PROGRAM PRG_HMI
VAR
	

	tonCaseDelay				: ARRAY [1..20] OF TON;
	tofCase						: ARRAY [1..20] OF TOF;
	rtrigCaseTriger				: ARRAY [1..20] OF R_TRIG;

	tonResetStatistics			: TON;
	
	fbWritePersistentData		:FB_WritePersistentData;
	fWritePersistentData		: F_TRIG;
	
END_VAR

ACT_ScreensNamesSet();
ACT_Buttons();
ACT_TimTrig();
ACT_General();
ACT_SavePersistentVariables();

tonResetStatistics( IN := 	GVL_HMI_GLOBAL.aResetHeightSensorBadParts [1] 	OR
							GVL_HMI_GLOBAL.aResetHeightSensorBadParts [2] 	OR
							GVL_HMI_GLOBAL.aResetHeightSensorBadParts [3] 	OR
							GVL_HMI_GLOBAL.aResetHeightSensorBadParts [4] 	OR
							GVL_HMI_GLOBAL.aResetHeightSensorGoodParts[1]	OR
							GVL_HMI_GLOBAL.aResetHeightSensorGoodParts[2]	OR
							GVL_HMI_GLOBAL.aResetHeightSensorGoodParts[3]	OR
							GVL_HMI_GLOBAL.aResetHeightSensorGoodParts[4]	OR
							GVL_HMI_GLOBAL.bResetHeightFailParts			OR
							GVL_HMI_GLOBAL.bResetHeightGoodParts			OR
							GVL_HMI_GLOBAL.bResetGoodParts					OR
							GVL_HMI_GLOBAL.bResetVisionBadParts				OR
							GVL_HMI_GLOBAL.bResetVisionGoodParts			OR
							GVL_HMI_GLOBAL.bResetFailedParts				OR
							GVL_HMI_GLOBAL.bResetGoodParts					,
							PT												:= T#500MS);

ACTION ACT_Buttons:
ACT_TimTrig();

IF tonCaseDelay[1].Q THEN
	
		GVL_HMI_GLOBAL.bResetButton	:= FALSE;
		
END_IF
IF tonCaseDelay[2].Q THEN
	
		GVL_HMI_GLOBAL.bStopButton	:= FALSE;
		
END_IF
IF tonCaseDelay[3].Q THEN
	
		GVL_HMI_GLOBAL.bStartButton	:= FALSE;
		
END_IF



IF tonCaseDelay[7].Q THEN
	
		GVL_HMI_GLOBAL.bShutDown	:= FALSE;
		
END_IF


IF tonCaseDelay[9].Q THEN
	
		GVL_HMI_GLOBAL.bSetSetPointsHeightTest	:= FALSE;
		
END_IF

IF tonCaseDelay[10].Q THEN
	
		GVL_HMI_GLOBAL.bManualMeasureHeightTest	:= FALSE;
		
END_IF

IF tonResetStatistics.Q THEN
	
							GVL_HMI_GLOBAL.aResetHeightSensorBadParts [1] 	:= FALSE;
							GVL_HMI_GLOBAL.aResetHeightSensorBadParts [2] 	:= FALSE;
							GVL_HMI_GLOBAL.aResetHeightSensorBadParts [3] 	:= FALSE;
							GVL_HMI_GLOBAL.aResetHeightSensorBadParts [4] 	:= FALSE;
							GVL_HMI_GLOBAL.aResetHeightSensorGoodParts[1]	:= FALSE;
							GVL_HMI_GLOBAL.aResetHeightSensorGoodParts[2]	:= FALSE;
							GVL_HMI_GLOBAL.aResetHeightSensorGoodParts[3]	:= FALSE;
							GVL_HMI_GLOBAL.aResetHeightSensorGoodParts[4]	:= FALSE;
							GVL_HMI_GLOBAL.bResetHeightFailParts			:= FALSE;
							GVL_HMI_GLOBAL.bResetHeightGoodParts			:= FALSE;
							GVL_HMI_GLOBAL.bResetGoodParts					:= FALSE;
							GVL_HMI_GLOBAL.bResetVisionBadParts				:= FALSE;
							GVL_HMI_GLOBAL.bResetVisionGoodParts			:= FALSE;
							GVL_HMI_GLOBAL.bResetFailedParts				:= FALSE;
							GVL_HMI_GLOBAL.bResetGoodParts					:= FALSE;


END_IF
END_ACTION

ACTION ACT_General:
IF tofCase[1].Q AND 
( NOT GVL_MASTER.stMasterControl.bNoStationImmediateFault OR NOT GVL_MASTER.stMasterControl.bNoCycleStopFault) THEN
	GVL_HMI_GLOBAL.bAutocycleFaultDialog := TRUE;
END_IF
END_ACTION

ACTION ACT_SavePersistentVariables:
fWritePersistentData(CLK := GVL_HMI_GLOBAL.nRegionMain = 5);

fbWritePersistentData(	PORT 				:= 851,
						START 				:= fWritePersistentData.Q,);
END_ACTION

ACTION ACT_ScreensNamesSet:
GVL_HMI_GLOBAL.aIOScreen[0] := 'Overview';
GVL_HMI_GLOBAL.aIOScreen[1] := 'HMI - CP2913-0000 | Beckhoff HMI';
GVL_HMI_GLOBAL.aIOScreen[2] := 'PLC - C6015-0010 | Beckhoff PLC | Windows 10 Embedded';
GVL_HMI_GLOBAL.aIOScreen[3] := 'Terminal 1- EK1100 | EtherCAT Coupler';
GVL_HMI_GLOBAL.aIOScreen[4] := 'Terminal 2 - EL6070 | Licence ';
GVL_HMI_GLOBAL.aIOScreen[5] := CONCAT('Terminal 3 - ' , GVL_IO.dw_T02_EL1809.sTerminalName);
GVL_HMI_GLOBAL.aIOScreen[6] := CONCAT('Terminal 4 - ' , GVL_IO.dw_T03_EL2809.sTerminalName);
GVL_HMI_GLOBAL.aIOScreen[7] := 'Terminal 12 - EL6631 |  2-port communication interface';
GVL_HMI_GLOBAL.aIOScreen[8] := 'DL-PN1 4Keyence Communication Unit | IV4 Camera | ProfiNET';


GVL_HMI_GLOBAL.aManualScreen[0] := 'Keyence | Vision Test';
GVL_HMI_GLOBAL.aManualScreen[1] := 'Keyence | Height Test';
END_ACTION

ACTION ACT_TimTrig:


tonCaseDelay[1](IN:= GVL_HMI_GLOBAL.bResetButton,PT:=T#500MS);
tonCaseDelay[2](IN:= GVL_HMI_GLOBAL.bStopButton,PT:=T#500MS);
tonCaseDelay[3](IN:= GVL_HMI_GLOBAL.bStartButton,PT:=T#500MS);
tonCaseDelay[4](IN:= ,PT:=T#500MS);
tonCaseDelay[5](IN:= ,PT:=T#500MS);
tonCaseDelay[6](IN:= ,PT:=T#500MS);
//tonCaseDelay[7](IN:= GVL_HMI_GLOBAL.bShutDown,PT:=T#500MS);
tonCaseDelay[8](IN:= ,PT:=T#5S);
tonCaseDelay[9](IN:= GVL_HMI_GLOBAL.bSetSetPointsHeightTest,PT:=T#1S);
tonCaseDelay[10](IN:= GVL_HMI_GLOBAL.bManualMeasureHeightTest,PT:=T#1S);

tofCase[1](IN:= (GVL_Master.stStationSruct[0].nState > 1000 AND GVL_Master.stStationSruct[0].nState < 1900),PT:=T#1S);


rtrigCaseTriger[1](CLK := GVL_MASTER.stNest.bPieceReject);
END_ACTION

END_PROGRAM

(* stored: Version 1.1.0.1, ProductVersion 3.1.4024.12
   POU PRG_HMI: Id {1fa80f95-1dd5-4aa8-847a-7b5565884994}, SpecialFunc None
   Action ACT_Buttons: Id {516d1fa4-b74a-4152-be9e-d2291d807b03}
   Action ACT_General: Id {435b764e-e0a8-4f56-b267-66ba0d9eee9f}
   Action ACT_SavePersistentVariables: Id {cefdb6b4-8666-42ec-915e-52d05413d6b5}
   Action ACT_ScreensNamesSet: Id {cfb190dc-badd-4760-9c94-186ee66d1d38}
   Action ACT_TimTrig: Id {c608156b-aba3-4ac2-9426-32de0bea0b69} *)
